TYPE ST_XMotionStatemachineStates :
STRUCT
	nAbortState		: INT;
	nResetState		: INT;
	nPrepareState	: INT;
	nStartState		: INT;
END_STRUCT
END_TYPE

(* stored: Version 1.1.0.1, ProductVersion 3.1.4024.4
   DUT ST_XMotionStatemachineStates: Id {306a63c8-78ad-4e66-9434-2ad4de3a59d4} *)
